% RSLogix 500 project RUTUJA1.RSS, saved by version 8.30.00.16 %
PROJECT "UNTITLED"    % processor: Bul.1763 MicroLogix 1100 Series B %

PROGRAM FILES
  LAD 2   7 rungs

DATA FILES
  O0 OUTPUT  4 elements
  I1 INPUT  6 elements
  S2 STATUS  66 elements
  B3 BINARY  1 elements
  T4 TIMER  1 elements
  C5 COUNTER  1 elements
  R6 CONTROL  1 elements
  N7 INTEGER  1 elements
  F8 FLOAT  1 elements

LADDER 2
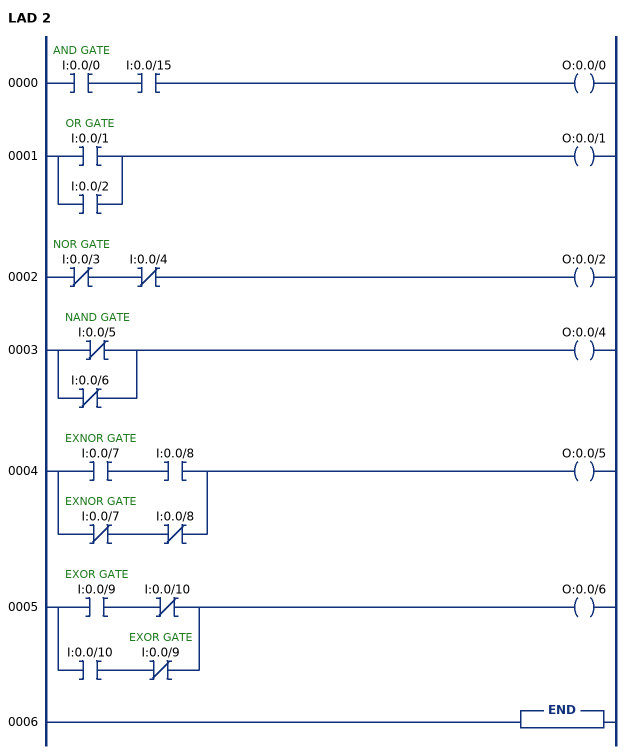
% Rung: 0 %
SOR XIC I:0.0/0 XIC I:0.0/15 OTE O:0.0/0 EOR
%   I:0.0/0  "AND GATE" %
% Rung: 1 %
SOR BST XIC I:0.0/1 NXB XIC I:0.0/2 BND OTE O:0.0/1 EOR
%   I:0.0/1  "OR GATE" %
% Rung: 2 %
SOR XIO I:0.0/3 XIO I:0.0/4 OTE O:0.0/2 EOR
%   I:0.0/3  "NOR GATE" %
% Rung: 3 %
SOR BST XIO I:0.0/5 NXB XIO I:0.0/6 BND OTE O:0.0/4 EOR
%   I:0.0/5  "NAND GATE" %
% Rung: 4 %
SOR BST XIC I:0.0/7 XIC I:0.0/8 NXB XIO I:0.0/7 XIO I:0.0/8 BND OTE O:0.0/5 EOR
%   I:0.0/7  "EXNOR GATE" %
% Rung: 5 %
SOR BST XIC I:0.0/9 XIO I:0.0/10 NXB XIC I:0.0/10 XIO I:0.0/9 BND OTE O:0.0/6 EOR
%   I:0.0/9  "EXOR GATE" %
% Rung: 6 %
SOR END EOR
